// Mitsubishi GX Works2 project: a15   PLC: Q02/Q02H

PROGRAM MAIN
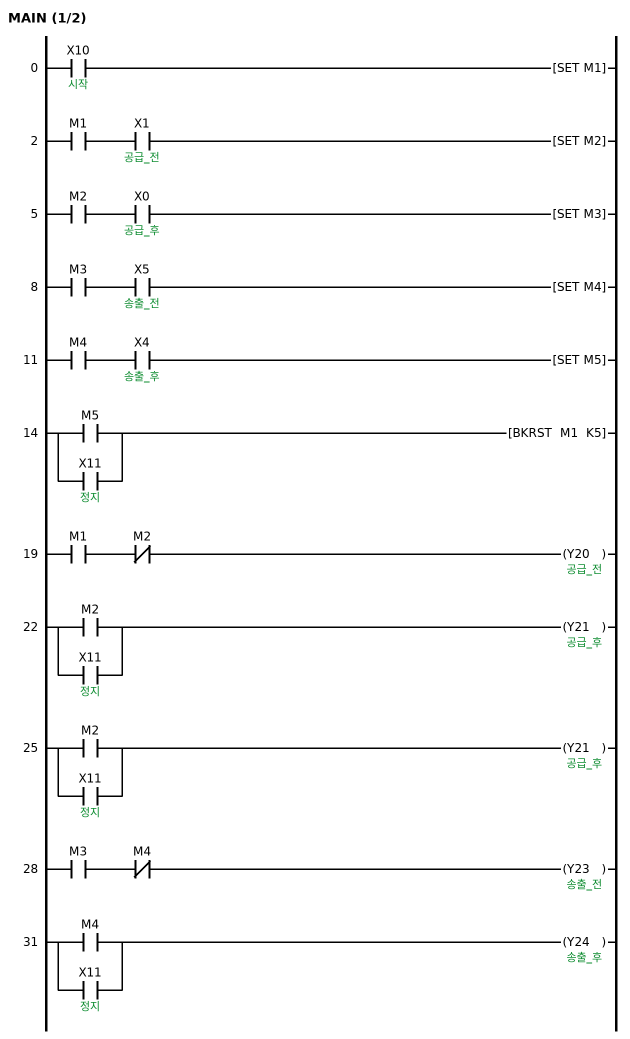
0     LD      X10  ; 시작
      SET     M1
2     LD      M1
      AND     X1  ; 공급_전
      SET     M2
5     LD      M2
      AND     X0  ; 공급_후
      SET     M3
8     LD      M3
      AND     X5  ; 송출_전
      SET     M4
11    LD      M4
      AND     X4  ; 송출_후
      SET     M5
14    LD      M5
      OR      X11  ; 정지
      BKRST   M1 K5
19    LD      M1
      ANI     M2
      OUT     Y20  ; 공급_전
22    LD      M2
      OR      X11  ; 정지
      OUT     Y21  ; 공급_후
25    LD      M2
      OR      X11  ; 정지
      OUT     Y21  ; 공급_후
28    LD      M3
      ANI     M4
      OUT     Y23  ; 송출_전
31    LD      M4
      OR      X11  ; 정지
      OUT     Y24  ; 송출_후
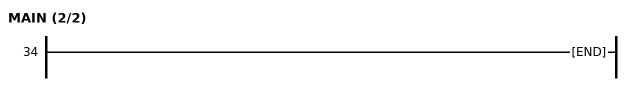
34    END
END_PROGRAM

// device comments not shown above
X2  ; 드릴_상
X3  ; 드릴_하
X6  ; 배출_후
X7  ; 배출_전
Y22  ; 드릴_하
Y25  ; 배출_전
Y26  ; 배출_후
Y29  ; RL
Y2A  ; YL
Y2B  ; GL
